(* Logix 5000 project; controller DUNEW2PLC1 vendor 1 type 14 code 221 rev 33.11; software revision 33.00; part 3 of 4 *)
(* tags used below, declared in another part *)
   accel_xy : REAL;   // Tangential acceleration of the winding head in xy-plane
   ACTUATOR_POS : DINT;
   ALL_EOT_GOOD : BOOL;
   APA_IS_VERTICAL : BOOL;
   check_tension_stable : BOOL;   // Check if the tension is stable at the setpoint before moving the winding head
   current_command : REAL;
   current_command_high : REAL;
   current_command_low : REAL;
   ERROR_CODE : DINT;
   gamma : REAL;
   J : REAL;
   LATCH_ACTUATOR_HOMED : BOOL;
   MAS : BOOL;   // Motion Axis Stop
   MASTER_Z_GO : BOOL;
   max_tolerable_tension : REAL;
   MAX_TOLERABLE_Z : REAL;
   MCCD_X_Y_Axis : MOTION_INSTRUCTION;
   MCCD_X_Y_Axis1 : MOTION_INSTRUCTION;
   MORE_STATS : BOOL[32];
   MOVE_TYPE : INT;   // 0 = No Move 1 = XY JOG 2 = XY Plane Move 3 = Z JOG 4 = Z Axis Move 5 = Toggle Latch Actuator 6 = Home the Latch Actuator
   neutral_cv : REAL;
   NEXTSTATE : DINT;
   overtension_timer : TIMER;
   pid_cv_high_limit : REAL;
   pid_cv_low_limit : REAL;
   pid_cv_out : REAL;
   PID_LOOP_TIMER : TIMER;
   pid_loop_timer_bypass : BOOL;
   Safety_Tripped_S : BOOL;
   SetPoint_CV : REAL;
   SetPoint_Override : REAL;
   SetPoint_PV : REAL;   // wire tension from load cell (N)
   SLS_speed : DINT;
   speed_regulator_switch : BOOL;   // This is our "enable safe speed" switch, repurposed to switch the speed regulator
   STATE : DINT;   // CURRENT State Machine State
   tension : ALIAS FOR Local:4:I.Ch01.Data;   // wire tension (N)
   TENSION_CONTROL_OK : BOOL;
   TENSION_ON_SWITCH : BOOL;
   tension_on_switch_delay_on_start : TIMER;
   tension_setpoint : REAL;
   tension_stable_timer : TIMER;
   v_0 : REAL;
   v_xyz : REAL;   // Velocity of winding head in xyz space
   winding_head_pid : PID;
   wire_break_proxy : BOOL;
   X_axis : AXIS_CIP_DRIVE;
   X_Axis_SLS : SAFELY_LIMITED_SPEED;
   X_POSITION : ALIAS FOR POSITION[0,0];
   X_Y : COORDINATE_SYSTEM;
   XY_ACCELERATION : REAL;   // Maximum positive acceleration for position move.
   XY_DECELERATION : REAL;   // Maximum negative acceleration for position move.
   XY_DECELERATION_SLS : REAL;
   xy_regulated_acceleration : REAL;
   xy_regulated_deceleration : REAL;
   XY_SPEED : REAL;   // Maximum velocity for position move.
   XY_SPEED_REQ : REAL;   // XY Requested speed copy of XY_Speed to be used for MCLM and MCCD in MoveXY
   Y_axis : AXIS_CIP_DRIVE;
   Y_POSITION : ALIAS FOR POSITION[0,1];
   Z_ACCELERATION : REAL;
   Z_axis : AXIS_CIP_DRIVE;
   Z_DECELLERATION : REAL;
   Z_FIXED_LATCHED : BOOL;
   Z_POSITION : REAL;
   Z_RETRACTED : BOOL;
   Z_SPEED : REAL;

PROGRAM MoveXY_State_2_3   (* main routine MoveXY *)
VAR
   d_raw : REAL;
   dx : REAL := 0.0039;
   dy : REAL := 0.0017;
   eot_triggered : BOOL;
   k : REAL := 211538.47;
   max_integral : DINT := 1000;
   min_integral : DINT := -1000;
   min_regulated_speed : DINT := 100;
   near_ending : BOOL;   // True if distance to xy-move target is less than the required stopping distance
   near_ending_trigger : BOOL;
   oneshotob : BOOL[32];
   oneshotsb : BOOL[32] := ([2] := 1, [4] := 1, [11] := 1, [12] := 1, [13] := 1, [14] := 1, [15] := 1, [16] := 1, [17] := 1);
   regulated_speed : REAL := 899.9713;
   regulator_loop_timer : TIMER := (PRE := 1);
   speed_set_to_zero : BOOL;
   speed_tension_setpoint : REAL := 8.5;
   starting_x : REAL := -0.0039;
   starting_y : REAL := -0.0017;
   STATE3_IND : BOOL; {access Read Only}
   stopping_distance : REAL;   // Calculate the distance required to perform a jerk-limited stop at the gurrent jerk, acceleration, and speed
   stopping_ratio : REAL := 0.2532453;
   trigger_xy_move : BOOL;
   v_max : REAL := 899.9713;
   x_dist_to_target : REAL := 0.6653;
   X_max_speed : REAL := 825.0; {constant}
   x_time : REAL := 211538.47;
   xy_accel_jerk : DINT := 1500;
   XY_AXIS_STAT : MOTION_INSTRUCTION[32] := ([2].FLAGS := 536870912, [2].DN := 1, [3].FLAGS := 536870912, [3].DN := 1, [4].FLAGS := 33554432, [5].FLAGS := 33554432, [6].FLAGS := 704643072, [6].DN := 1, [6].PC := 1);
   xy_d_alpha : REAL := 1.0;
   xy_d_dt : DINT := 50;
   xy_d_term : REAL;
   xy_d_term_prev : REAL;
   xy_d_timer : TIMER := (PRE := 50);
   xy_decel_jerk : DINT := 2000;
   xy_default_speed : DINT;
   xy_dist_to_target : REAL := 0.66530246;
   xy_dt : DINT := 1;
   xy_error : REAL := 6.0954127;
   xy_error_prev : REAL := 6.0985594;
   xy_i_term : REAL := 900.0352;
   xy_kd : REAL;
   xy_ki : REAL := 300.0;
   xy_kp : REAL;
   xy_p_term : REAL;
   XY_POS_LOCK_STAT : BOOL; {access Read Only}
   y_dist_to_target : REAL := -0.0018;
   Y_max_speed : REAL := 600.0; {constant}
   y_time : REAL := 352941.16;
END_VAR

ROUTINE MoveXY   (* ladder *)
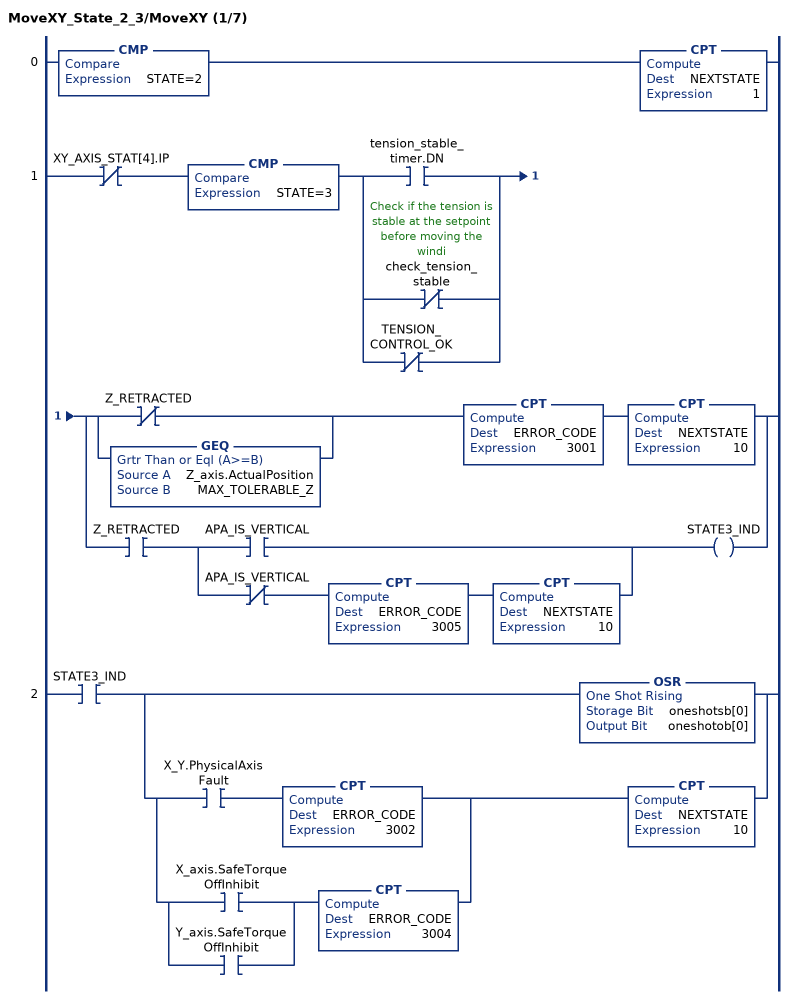
   0: CMP(STATE=2)CPT(NEXTSTATE,1);
   1: XIO(XY_AXIS_STAT[4].IP)CMP(STATE=3)[XIC(tension_stable_timer.DN) ,XIO(check_tension_stable) ,XIO(TENSION_CONTROL_OK) ][[XIO(Z_RETRACTED) ,GEQ(Z_axis.ActualPosition,MAX_TOLERABLE_Z) ] CPT(ERROR_CODE,3001) CPT(NEXTSTATE,10) ,XIC(Z_RETRACTED) [XIC(APA_IS_VERTICAL) ,XIO(APA_IS_VERTICAL) CPT(ERROR_CODE,3005) CPT(NEXTSTATE,10) ] OTE(STATE3_IND) ];
   2: XIC(STATE3_IND)[OSR(oneshotsb[0],oneshotob[0]) ,[XIC(X_Y.PhysicalAxisFault) CPT(ERROR_CODE,3002) ,[XIC(X_axis.SafeTorqueOffInhibit) ,XIC(Y_axis.SafeTorqueOffInhibit) ] CPT(ERROR_CODE,3004) ] CPT(NEXTSTATE,10) ];
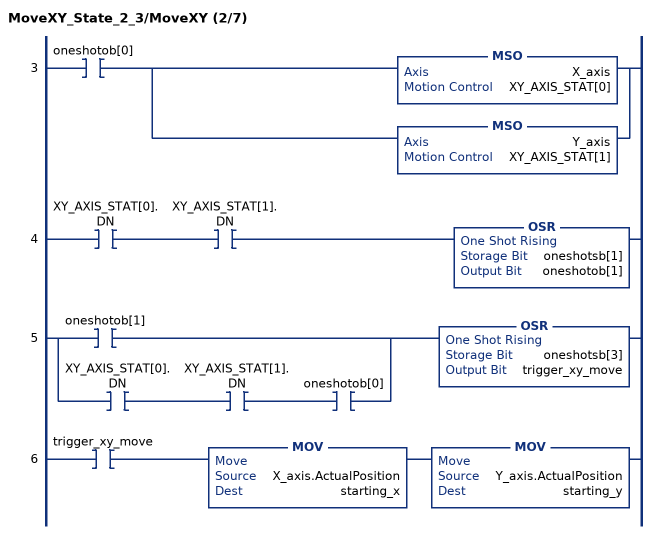
   3: XIC(oneshotob[0])[MSO(X_axis,XY_AXIS_STAT[0]) ,MSO(Y_axis,XY_AXIS_STAT[1]) ];
   4: XIC(XY_AXIS_STAT[0].DN)XIC(XY_AXIS_STAT[1].DN)OSR(oneshotsb[1],oneshotob[1]);
   5: [XIC(oneshotob[1]) ,XIC(XY_AXIS_STAT[0].DN) XIC(XY_AXIS_STAT[1].DN) XIC(oneshotob[0]) ]OSR(oneshotsb[3],trigger_xy_move);
   6: XIC(trigger_xy_move)MOV(X_axis.ActualPosition,starting_x)MOV(Y_axis.ActualPosition,starting_y);
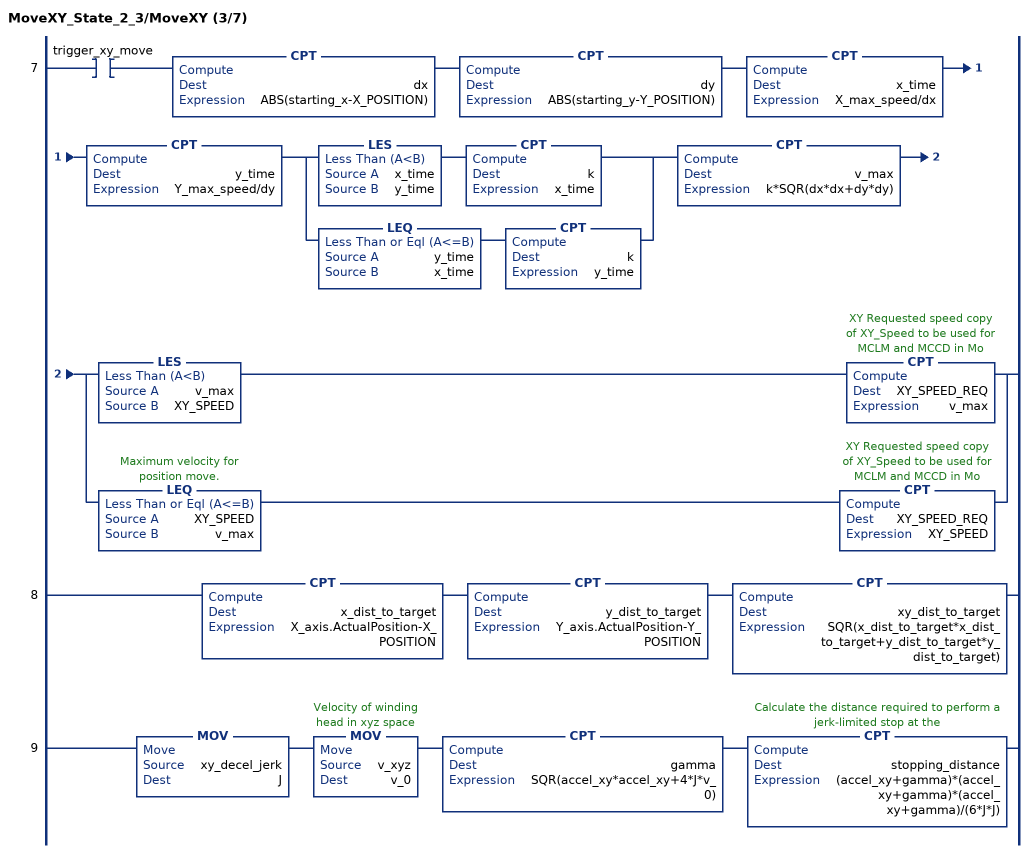
   7: XIC(trigger_xy_move)CPT(dx,ABS(starting_x-X_POSITION))CPT(dy,ABS(starting_y-Y_POSITION))CPT(x_time,X_max_speed/dx)CPT(y_time,Y_max_speed/dy)[LES(x_time,y_time) CPT(k,x_time) ,LEQ(y_time,x_time) CPT(k,y_time) ]CPT(v_max,k*SQR(dx*dx+dy*dy))[LES(v_max,XY_SPEED) CPT(XY_SPEED_REQ,v_max) ,LEQ(XY_SPEED,v_max) CPT(XY_SPEED_REQ,XY_SPEED) ];
   8: CPT(x_dist_to_target,X_axis.ActualPosition-X_POSITION)CPT(y_dist_to_target,Y_axis.ActualPosition-Y_POSITION)CPT(xy_dist_to_target,SQR(x_dist_to_target*x_dist_to_target+y_dist_to_target*y_dist_to_target));
   9: MOV(xy_decel_jerk,J)MOV(v_xyz,v_0)CPT(gamma,SQR(accel_xy*accel_xy+4*J*v_0))CPT(stopping_distance,(accel_xy+gamma)*(accel_xy+gamma)*(accel_xy+gamma)/(6*J*J));
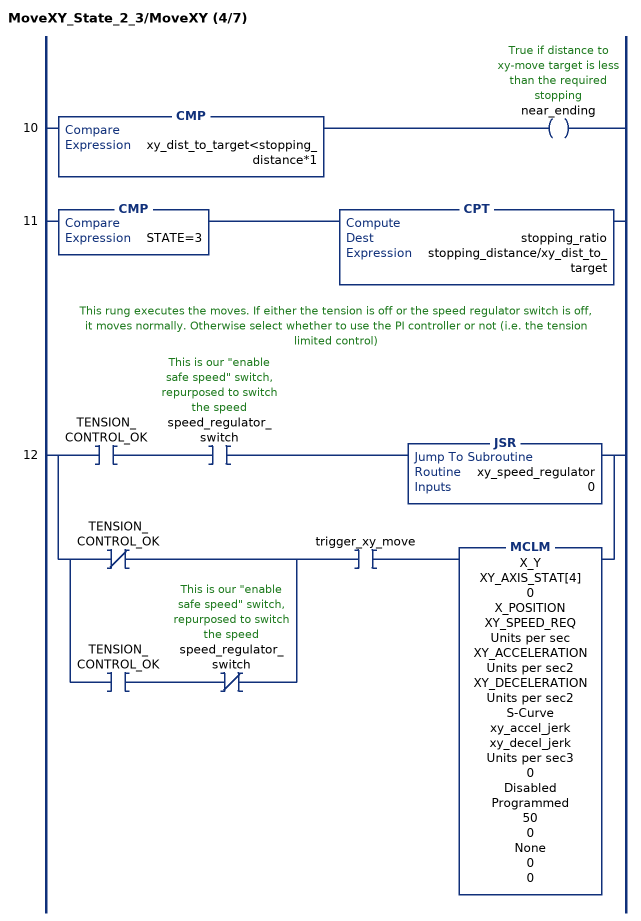
   10: CMP(xy_dist_to_target<stopping_distance*1)OTE(near_ending);
   11: CMP(STATE=3)CPT(stopping_ratio,stopping_distance/xy_dist_to_target);
   // This rung executes the moves. If either the tension is off or the speed regulator switch is off, it moves normally. Otherwise select whether to use the PI controller or not (i.e. the tension limited control)
   12: [XIC(TENSION_CONTROL_OK) XIC(speed_regulator_switch) JSR(xy_speed_regulator,0) ,[XIO(TENSION_CONTROL_OK) ,XIC(TENSION_CONTROL_OK) XIO(speed_regulator_switch) ] XIC(trigger_xy_move) MCLM(X_Y,XY_AXIS_STAT[4],0,X_POSITION,XY_SPEED_REQ,Units per sec,XY_ACCELERATION,Units per sec2,XY_DECELERATION,Units per sec2,S-Curve,xy_accel_jerk,xy_decel_jerk,Units per sec3,0,Disabled,Programmed,50,0,None,0,0) ];
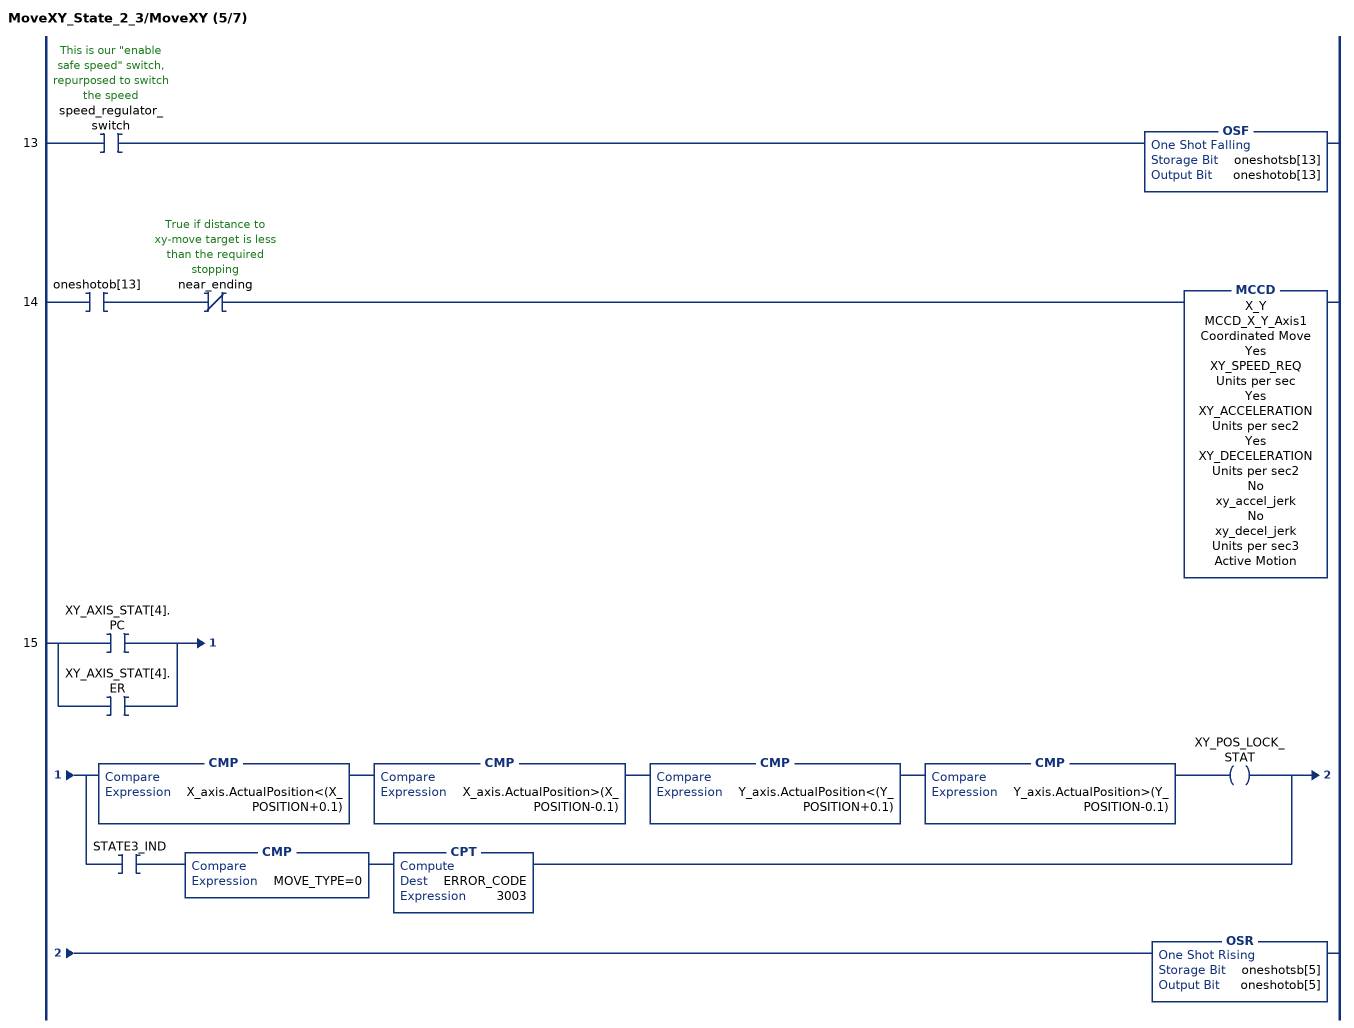
   13: XIC(speed_regulator_switch)OSF(oneshotsb[13],oneshotob[13]);
   14: XIC(oneshotob[13])XIO(near_ending)MCCD(X_Y,MCCD_X_Y_Axis1,Coordinated Move,Yes,XY_SPEED_REQ,Units per sec,Yes,XY_ACCELERATION,Units per sec2,Yes,XY_DECELERATION,Units per sec2,No,xy_accel_jerk,No,xy_decel_jerk,Units per sec3,Active Motion);
   15: [XIC(XY_AXIS_STAT[4].PC) ,XIC(XY_AXIS_STAT[4].ER) ][CMP(X_axis.ActualPosition<(X_POSITION+0.1)) CMP(X_axis.ActualPosition>(X_POSITION-0.1)) CMP(Y_axis.ActualPosition<(Y_POSITION+0.1)) CMP(Y_axis.ActualPosition>(Y_POSITION-0.1)) OTE(XY_POS_LOCK_STAT) ,XIC(STATE3_IND) CMP(MOVE_TYPE=0) CPT(ERROR_CODE,3003) ]OSR(oneshotsb[5],oneshotob[5]);
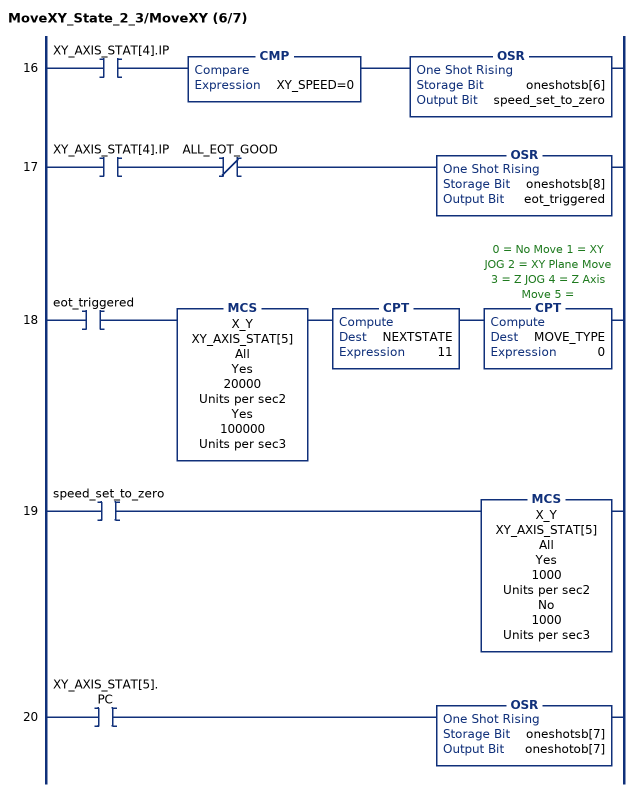
   16: XIC(XY_AXIS_STAT[4].IP)CMP(XY_SPEED=0)OSR(oneshotsb[6],speed_set_to_zero);
   17: XIC(XY_AXIS_STAT[4].IP)XIO(ALL_EOT_GOOD)OSR(oneshotsb[8],eot_triggered);
   18: XIC(eot_triggered)MCS(X_Y,XY_AXIS_STAT[5],All,Yes,20000,Units per sec2,Yes,100000,Units per sec3)CPT(NEXTSTATE,11)CPT(MOVE_TYPE,0);
   19: XIC(speed_set_to_zero)MCS(X_Y,XY_AXIS_STAT[5],All,Yes,1000,Units per sec2,No,1000,Units per sec3);
   20: XIC(XY_AXIS_STAT[5].PC)OSR(oneshotsb[7],oneshotob[7]);
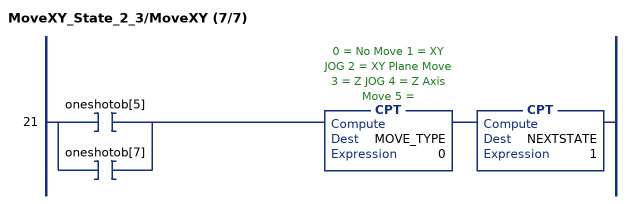
   21: [XIC(oneshotob[5]) ,XIC(oneshotob[7]) ]CPT(MOVE_TYPE,0)CPT(NEXTSTATE,1);
END_ROUTINE

ROUTINE xy_speed_regulator   (* ladder *)
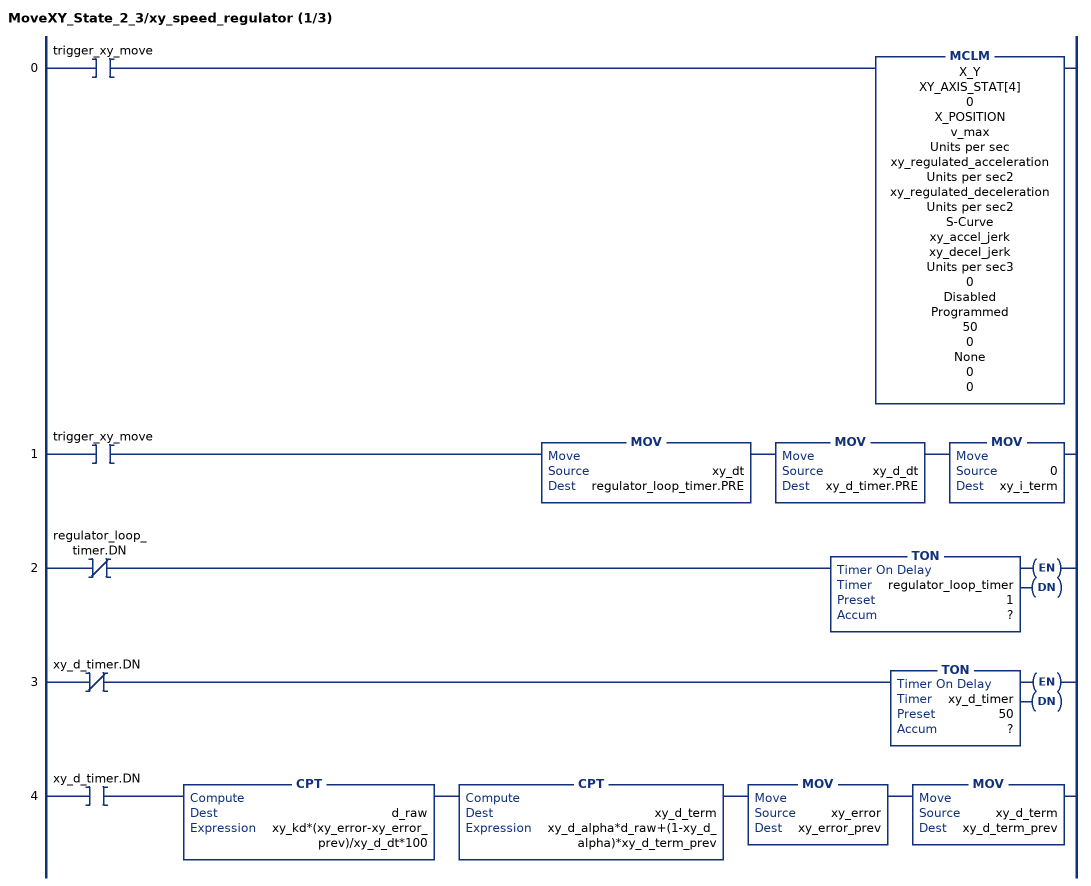
   0: XIC(trigger_xy_move)MCLM(X_Y,XY_AXIS_STAT[4],0,X_POSITION,v_max,Units per sec,xy_regulated_acceleration,Units per sec2,xy_regulated_deceleration,Units per sec2,S-Curve,xy_accel_jerk,xy_decel_jerk,Units per sec3,0,Disabled,Programmed,50,0,None,0,0);
   1: XIC(trigger_xy_move)MOV(xy_dt,regulator_loop_timer.PRE)MOV(xy_d_dt,xy_d_timer.PRE)MOV(0,xy_i_term);
   2: XIO(regulator_loop_timer.DN)TON(regulator_loop_timer,?,?);
   3: XIO(xy_d_timer.DN)TON(xy_d_timer,?,?);
   4: XIC(xy_d_timer.DN)CPT(d_raw,xy_kd*(xy_error-xy_error_prev)/xy_d_dt*100)CPT(xy_d_term,xy_d_alpha*d_raw+(1-xy_d_alpha)*xy_d_term_prev)MOV(xy_error,xy_error_prev)MOV(xy_d_term,xy_d_term_prev);
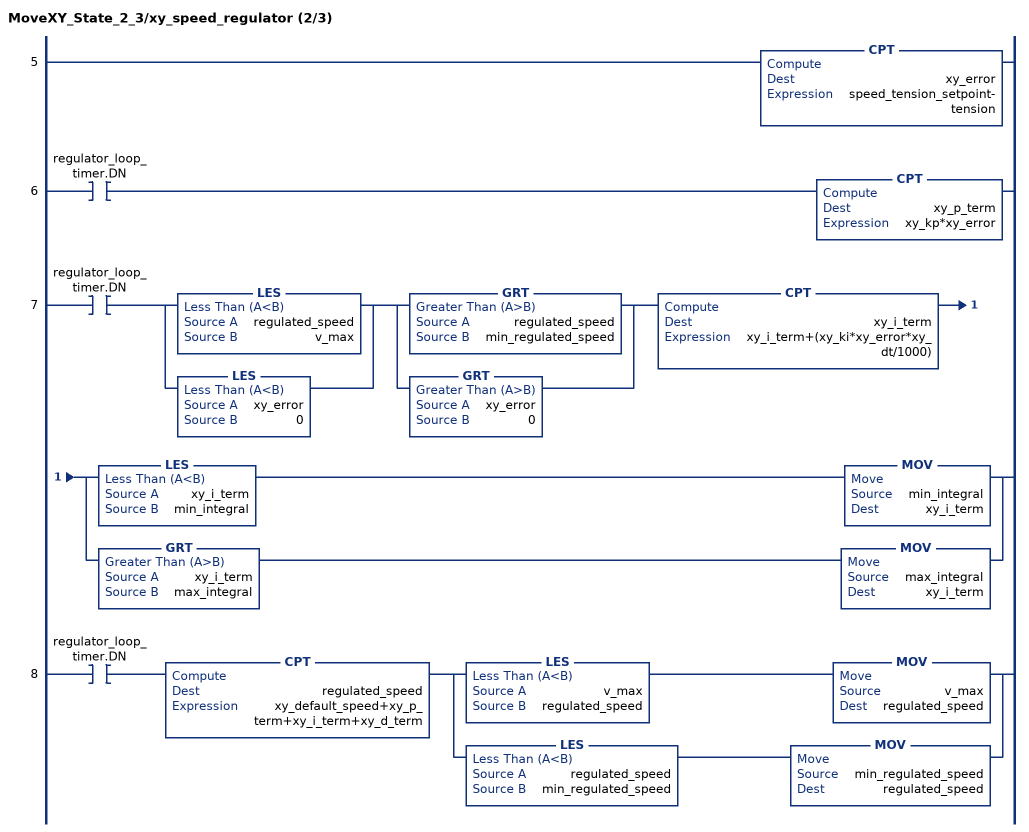
   5: CPT(xy_error,speed_tension_setpoint-tension);
   6: XIC(regulator_loop_timer.DN)CPT(xy_p_term,xy_kp*xy_error);
   7: XIC(regulator_loop_timer.DN)[LES(regulated_speed,v_max) ,LES(xy_error,0) ][GRT(regulated_speed,min_regulated_speed) ,GRT(xy_error,0) ]CPT(xy_i_term,xy_i_term+(xy_ki*xy_error*xy_dt/1000))[LES(xy_i_term,min_integral) MOV(min_integral,xy_i_term) ,GRT(xy_i_term,max_integral) MOV(max_integral,xy_i_term) ];
   8: XIC(regulator_loop_timer.DN)CPT(regulated_speed,xy_default_speed+xy_p_term+xy_i_term+xy_d_term)[LES(v_max,regulated_speed) MOV(v_max,regulated_speed) ,LES(regulated_speed,min_regulated_speed) MOV(min_regulated_speed,regulated_speed) ];
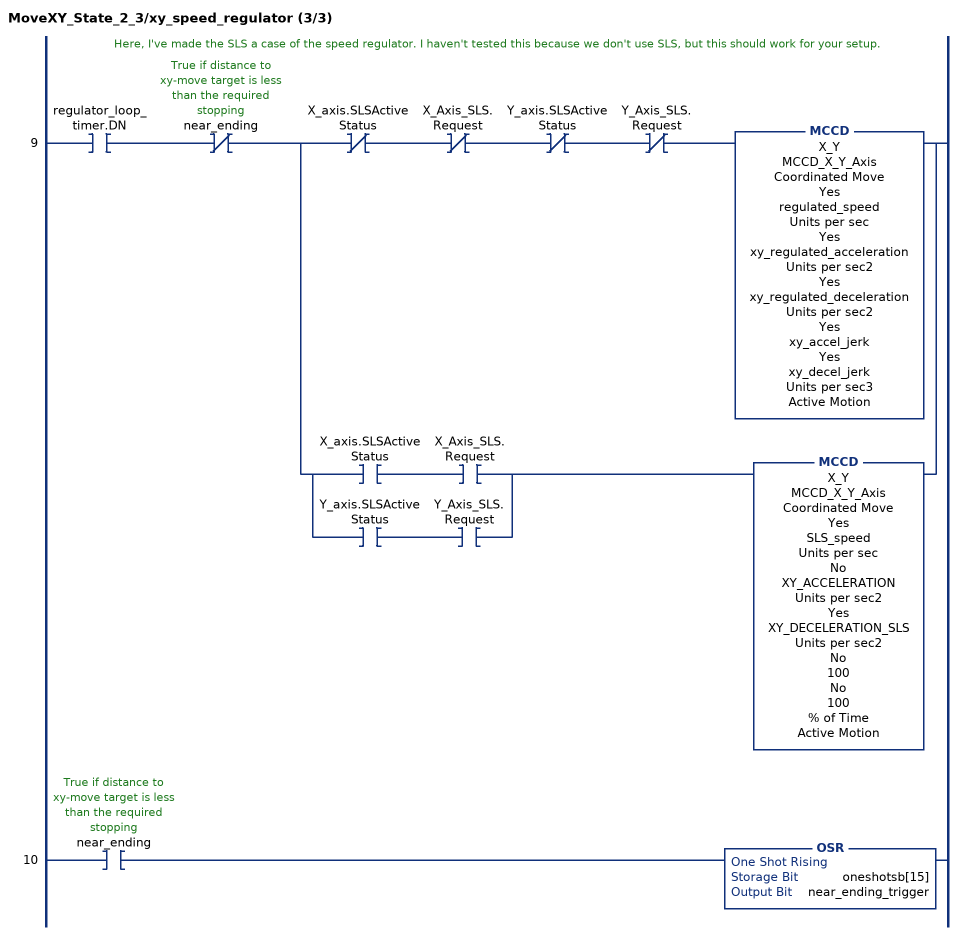
   // Here, I've made the SLS a case of the speed regulator. I haven't tested this because we don't use SLS, but this should work for your setup.
   9: XIC(regulator_loop_timer.DN)XIO(near_ending)[XIO(X_axis.SLSActiveStatus) XIO(X_Axis_SLS.Request) XIO(Y_axis.SLSActiveStatus) XIO(Y_Axis_SLS.Request) MCCD(X_Y,MCCD_X_Y_Axis,Coordinated Move,Yes,regulated_speed,Units per sec,Yes,xy_regulated_acceleration,Units per sec2,Yes,xy_regulated_deceleration,Units per sec2,Yes,xy_accel_jerk,Yes,xy_decel_jerk,Units per sec3,Active Motion) ,[XIC(X_axis.SLSActiveStatus) XIC(X_Axis_SLS.Request) ,XIC(Y_axis.SLSActiveStatus) XIC(Y_Axis_SLS.Request) ] MCCD(X_Y,MCCD_X_Y_Axis,Coordinated Move,Yes,SLS_speed,Units per sec,No,XY_ACCELERATION,Units per sec2,Yes,XY_DECELERATION_SLS,Units per sec2,No,100,No,100,% of Time,Active Motion) ];
   10: XIC(near_ending)OSR(oneshotsb[15],near_ending_trigger);
END_ROUTINE
END_PROGRAM

PROGRAM MoveZ_State_4_5   (* main routine MoveZ *)
VAR
   error_suppress : BOOL;
   oneshotob : BOOL[32]; {access Read Only}
   oneshotsb : BOOL[32] := ([0] := 1, [1] := 1, [2] := 1, [9] := 1, [26] := 1, [28] := 1, [29] := 1, [30] := 1, [31] := 1); {access Read Only}
   STATE5_IND : BOOL; {access Read Only}
   z_accel_jerk : DINT := 800;
   Z_AXIS_STAT : MOTION_INSTRUCTION[32] := ([0].FLAGS := 33554432, [1].FLAGS := 33554432, [2].FLAGS := 33554432, [4].FLAGS := 33554432, [5].FLAGS := 33554432, [6].FLAGS := 33554432, [7].FLAGS := 33554432, [8].FLAGS := 33554432, [9].FLAGS := 536870912, [9].DN := 1); {access Read Only}
   z_decel_jerk : DINT := 1600;
   Z_POS_LOCK_STAT : BOOL; {access Read Only}
END_VAR

ROUTINE MoveZ   (* ladder *)
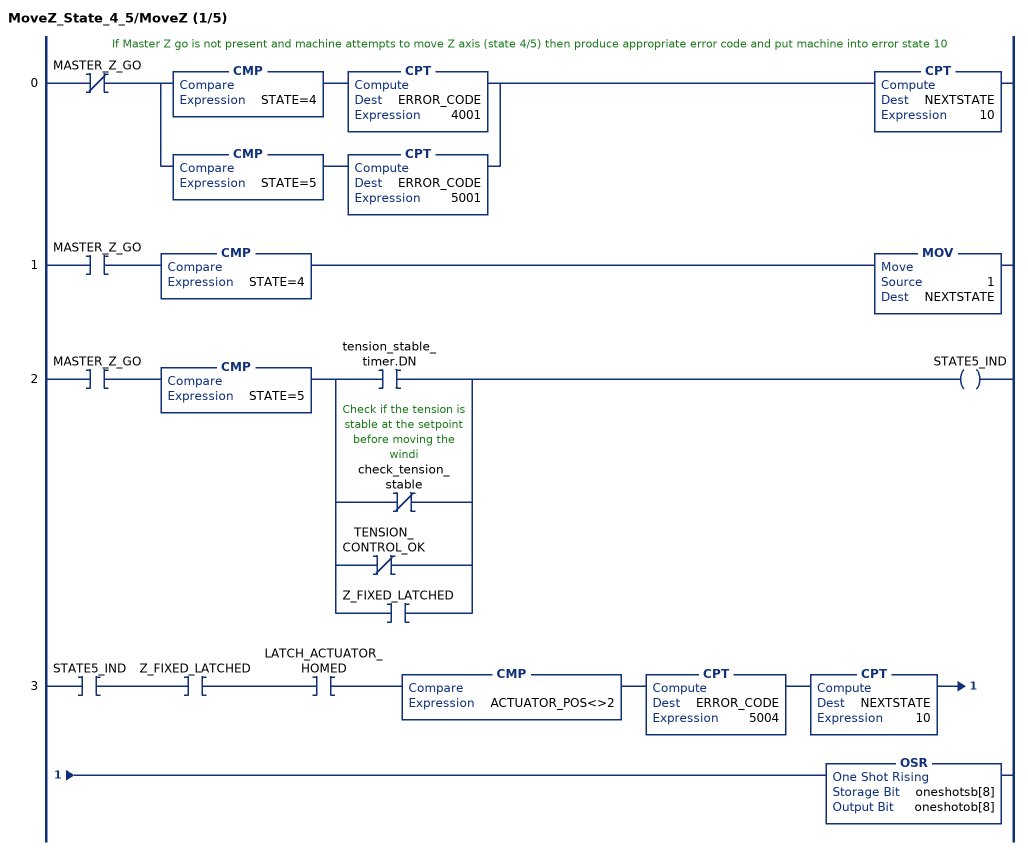
   // If Master Z go is not present and machine attempts to move Z axis (state 4/5) then produce appropriate error code and put machine into error state 10
   0: XIO(MASTER_Z_GO)[CMP(STATE=4) CPT(ERROR_CODE,4001) ,CMP(STATE=5) CPT(ERROR_CODE,5001) ]CPT(NEXTSTATE,10);
   1: XIC(MASTER_Z_GO)CMP(STATE=4)MOV(1,NEXTSTATE);
   2: XIC(MASTER_Z_GO)CMP(STATE=5)[XIC(tension_stable_timer.DN) ,XIO(check_tension_stable) ,XIO(TENSION_CONTROL_OK) ,XIC(Z_FIXED_LATCHED) ]OTE(STATE5_IND);
   3: XIC(STATE5_IND)XIC(Z_FIXED_LATCHED)XIC(LATCH_ACTUATOR_HOMED)CMP(ACTUATOR_POS<>2)CPT(ERROR_CODE,5004)CPT(NEXTSTATE,10)OSR(oneshotsb[8],oneshotob[8]);
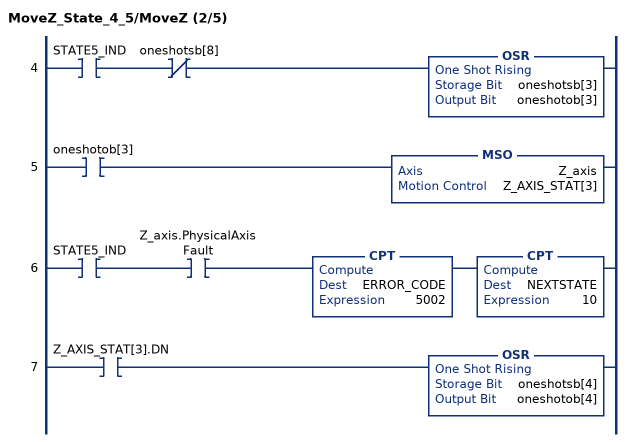
   4: XIC(STATE5_IND)XIO(oneshotsb[8])OSR(oneshotsb[3],oneshotob[3]);
   5: XIC(oneshotob[3])MSO(Z_axis,Z_AXIS_STAT[3]);
   6: XIC(STATE5_IND)XIC(Z_axis.PhysicalAxisFault)CPT(ERROR_CODE,5002)CPT(NEXTSTATE,10);
   7: XIC(Z_AXIS_STAT[3].DN)OSR(oneshotsb[4],oneshotob[4]);
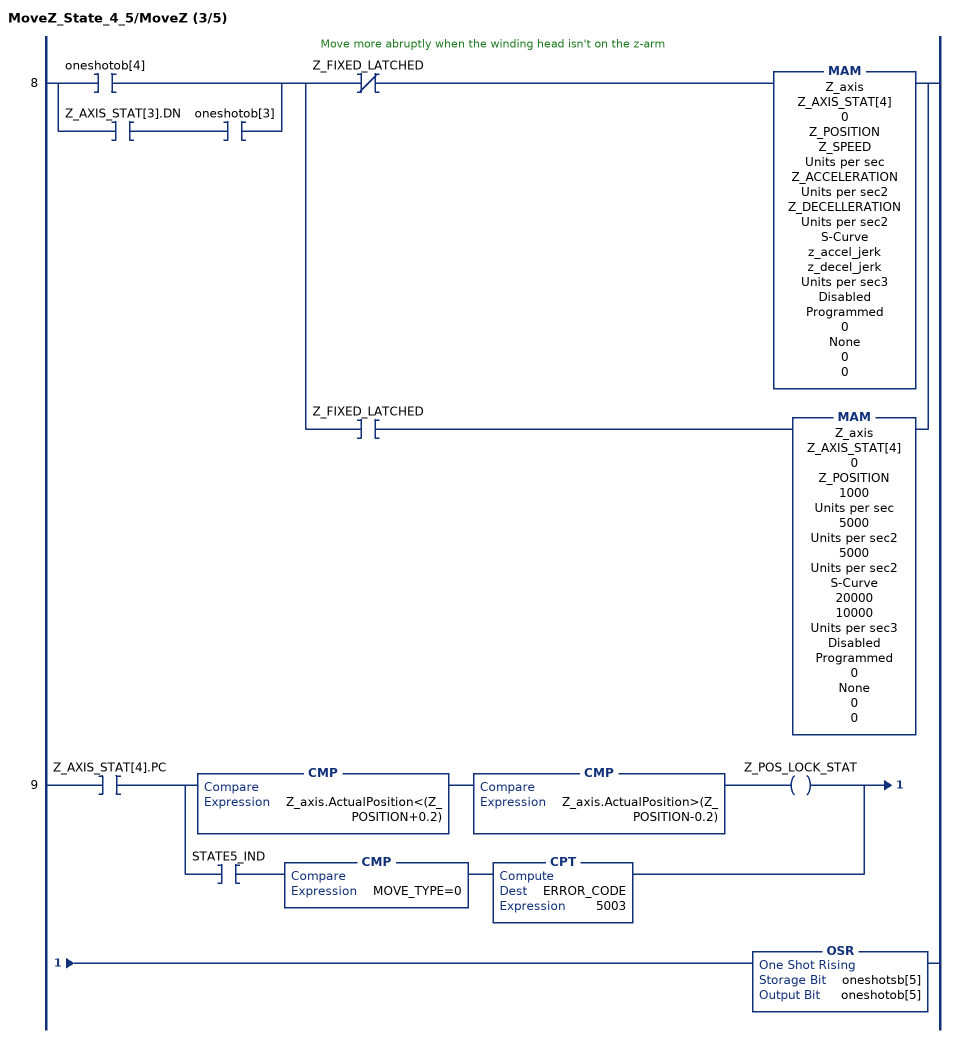
   // Move more abruptly when the winding head isn't on the z-arm
   8: [XIC(oneshotob[4]) ,XIC(Z_AXIS_STAT[3].DN) XIC(oneshotob[3]) ][XIO(Z_FIXED_LATCHED) MAM(Z_axis,Z_AXIS_STAT[4],0,Z_POSITION,Z_SPEED,Units per sec,Z_ACCELERATION,Units per sec2,Z_DECELLERATION,Units per sec2,S-Curve,z_accel_jerk,z_decel_jerk,Units per sec3,Disabled,Programmed,0,None,0,0) ,XIC(Z_FIXED_LATCHED) MAM(Z_axis,Z_AXIS_STAT[4],0,Z_POSITION,1000,Units per sec,5000,Units per sec2,5000,Units per sec2,S-Curve,20000,10000,Units per sec3,Disabled,Programmed,0,None,0,0) ];
   9: XIC(Z_AXIS_STAT[4].PC)[CMP(Z_axis.ActualPosition<(Z_POSITION+0.2)) CMP(Z_axis.ActualPosition>(Z_POSITION-0.2)) OTE(Z_POS_LOCK_STAT) ,XIC(STATE5_IND) CMP(MOVE_TYPE=0) CPT(ERROR_CODE,5003) ]OSR(oneshotsb[5],oneshotob[5]);
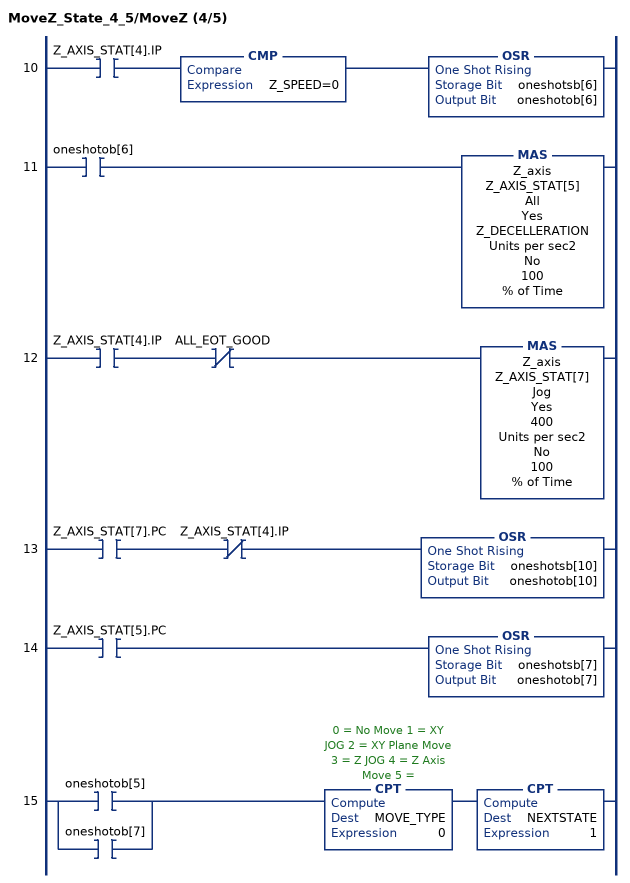
   10: XIC(Z_AXIS_STAT[4].IP)CMP(Z_SPEED=0)OSR(oneshotsb[6],oneshotob[6]);
   11: XIC(oneshotob[6])MAS(Z_axis,Z_AXIS_STAT[5],All,Yes,Z_DECELLERATION,Units per sec2,No,100,% of Time);
   12: XIC(Z_AXIS_STAT[4].IP)XIO(ALL_EOT_GOOD)MAS(Z_axis,Z_AXIS_STAT[7],Jog,Yes,400,Units per sec2,No,100,% of Time);
   13: XIC(Z_AXIS_STAT[7].PC)XIO(Z_AXIS_STAT[4].IP)OSR(oneshotsb[10],oneshotob[10]);
   14: XIC(Z_AXIS_STAT[5].PC)OSR(oneshotsb[7],oneshotob[7]);
   15: [XIC(oneshotob[5]) ,XIC(oneshotob[7]) ]CPT(MOVE_TYPE,0)CPT(NEXTSTATE,1);
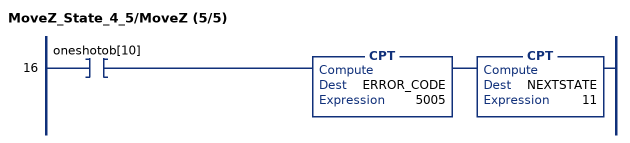
   16: XIC(oneshotob[10])CPT(ERROR_CODE,5005)CPT(NEXTSTATE,11);
END_ROUTINE
END_PROGRAM

PROGRAM PID_Tension_Servo   (* main routine PID_Tension *)
// Using code from Sarah Johnson
VAR
   constant_cv_out : BOOL;
   cv_to_electrocraft : ALIAS FOR Local:5:O.Ch00.Data;
   Enable_tension_motor : ALIAS FOR Local:3:O.Pt03.Data;
   oneshotob : BOOL[32];
   oneshotsb : BOOL[32];
   tension_stable_time : DINT := 200;
   tension_stable_tolerance : REAL := 0.15;
   wire_break_debounce : TIMER := (PRE := 50, ACC := 50, EN := 1, DN := 1);
   wire_break_switch_delay_on_start : TIMER := (PRE := 1000);
END_VAR

ROUTINE PID_Tension   (* ladder *)
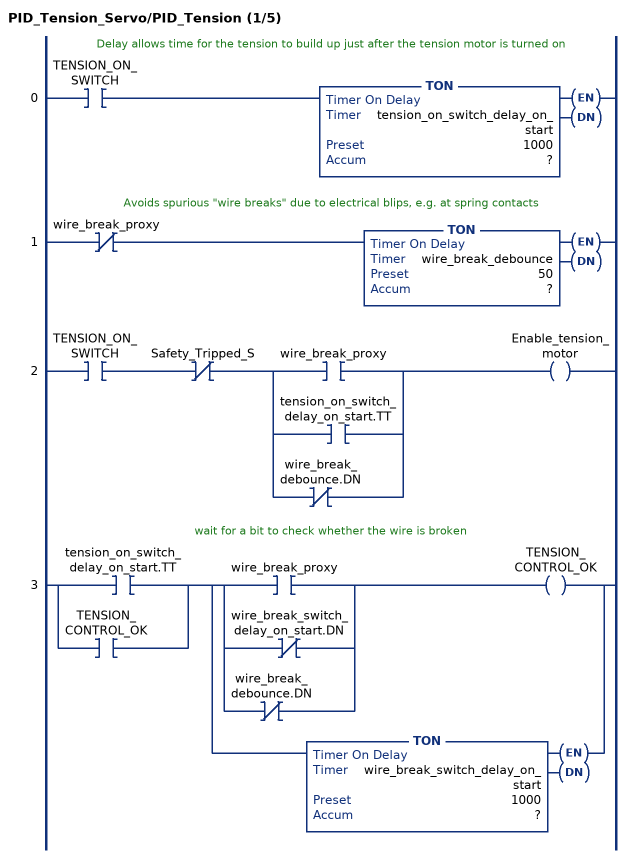
   // Delay allows time for the tension to build up just after the tension motor is turned on
   0: XIC(TENSION_ON_SWITCH)TON(tension_on_switch_delay_on_start,?,?);
   // Avoids spurious "wire breaks" due to electrical blips, e.g. at spring contacts
   1: XIO(wire_break_proxy)TON(wire_break_debounce,?,?);
   2: XIC(TENSION_ON_SWITCH)XIO(Safety_Tripped_S)[XIC(wire_break_proxy) ,XIC(tension_on_switch_delay_on_start.TT) ,XIO(wire_break_debounce.DN) ]OTE(Enable_tension_motor);
   // wait for a bit to check whether the wire is broken
   3: [XIC(tension_on_switch_delay_on_start.TT) ,XIC(TENSION_CONTROL_OK) ][[XIC(wire_break_proxy) ,XIO(wire_break_switch_delay_on_start.DN) ,XIO(wire_break_debounce.DN) ] OTE(TENSION_CONTROL_OK) ,TON(wire_break_switch_delay_on_start,?,?) ];
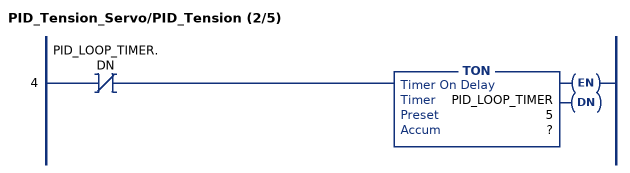
   4: XIO(PID_LOOP_TIMER.DN)TON(PID_LOOP_TIMER,?,?);
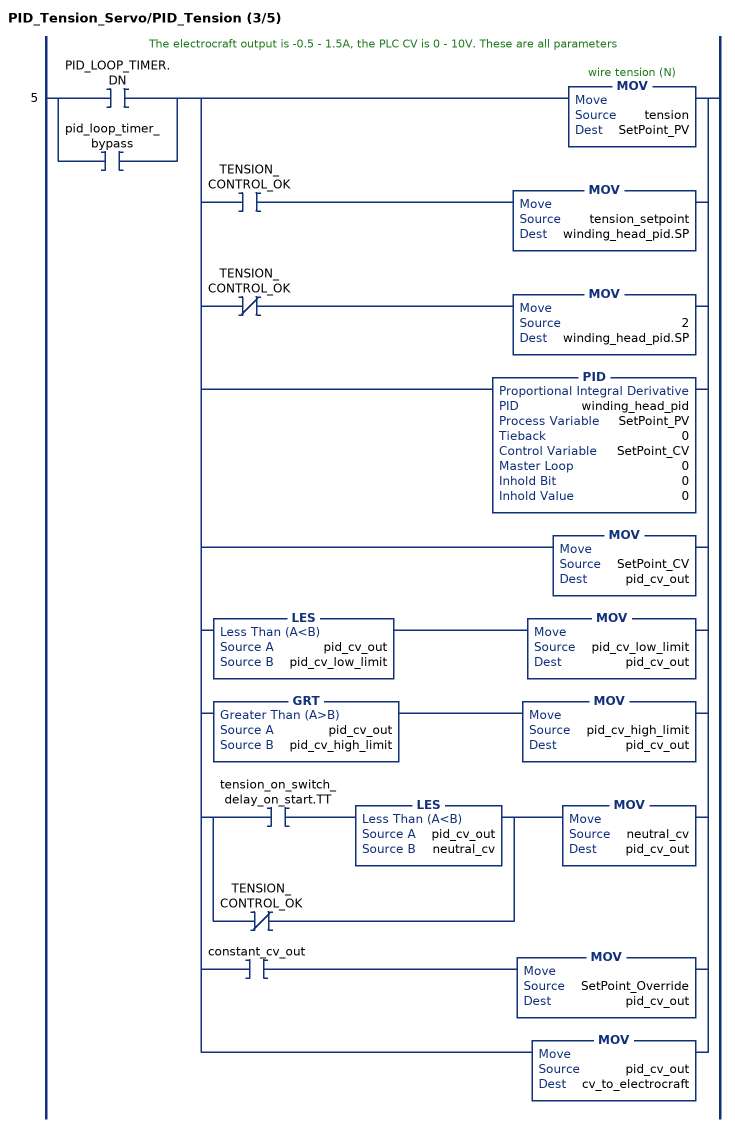
   // The electrocraft output is -0.5 - 1.5A, the PLC CV is 0 - 10V. These are all parameters
   5: [XIC(PID_LOOP_TIMER.DN) ,XIC(pid_loop_timer_bypass) ][MOV(tension,SetPoint_PV) ,XIC(TENSION_CONTROL_OK) MOV(tension_setpoint,winding_head_pid.SP) ,XIO(TENSION_CONTROL_OK) MOV(2,winding_head_pid.SP) ,PID(winding_head_pid,SetPoint_PV,0,SetPoint_CV,0,0,0) ,MOV(SetPoint_CV,pid_cv_out) ,LES(pid_cv_out,pid_cv_low_limit) MOV(pid_cv_low_limit,pid_cv_out) ,GRT(pid_cv_out,pid_cv_high_limit) MOV(pid_cv_high_limit,pid_cv_out) ,[XIC(tension_on_switch_delay_on_start.TT) LES(pid_cv_out,neutral_cv) ,XIO(TENSION_CONTROL_OK) ] MOV(neutral_cv,pid_cv_out) ,XIC(constant_cv_out) MOV(SetPoint_Override,pid_cv_out) ,MOV(pid_cv_out,cv_to_electrocraft) ];
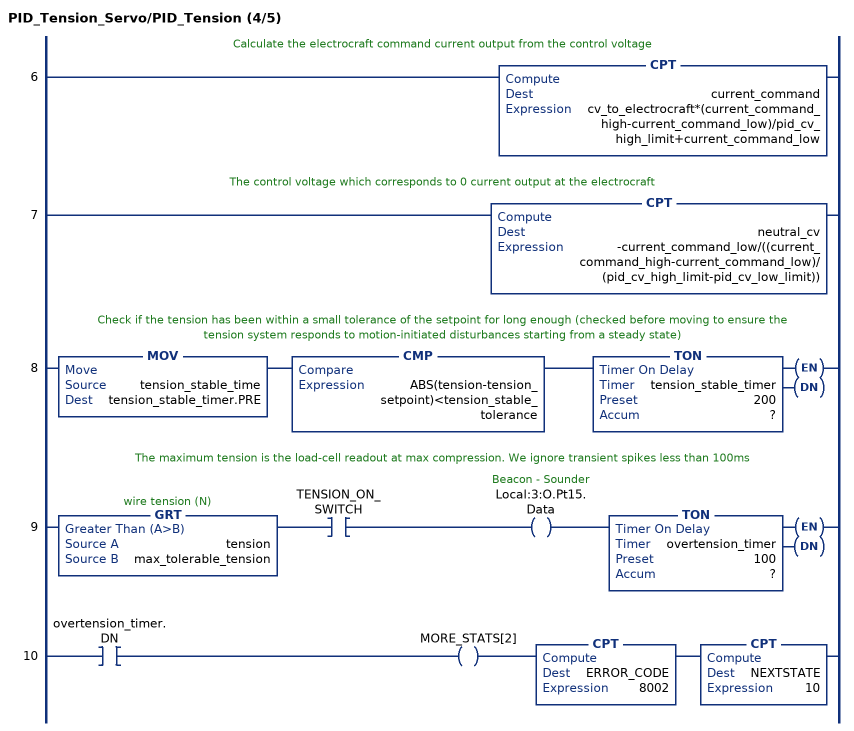
   // Calculate the electrocraft command current output from the control voltage
   6: CPT(current_command,cv_to_electrocraft*(current_command_high-current_command_low)/pid_cv_high_limit+current_command_low);
   // The control voltage which corresponds to 0 current output at the electrocraft
   7: CPT(neutral_cv,-current_command_low/((current_command_high-current_command_low)/(pid_cv_high_limit-pid_cv_low_limit)));
   // Check if the tension has been within a small tolerance of the setpoint for long enough (checked before moving to ensure the tension system responds to motion-initiated disturbances starting from a steady state)
   8: MOV(tension_stable_time,tension_stable_timer.PRE)CMP(ABS(tension-tension_setpoint)<tension_stable_tolerance)TON(tension_stable_timer,?,?);
   // The maximum tension is the load-cell readout at max compression. We ignore transient spikes less than 100ms
   9: GRT(tension,max_tolerable_tension)XIC(TENSION_ON_SWITCH)OTE(Local:3:O.Pt15.Data)TON(overtension_timer,?,?);
   10: XIC(overtension_timer.DN)OTE(MORE_STATS[2])CPT(ERROR_CODE,8002)CPT(NEXTSTATE,10);
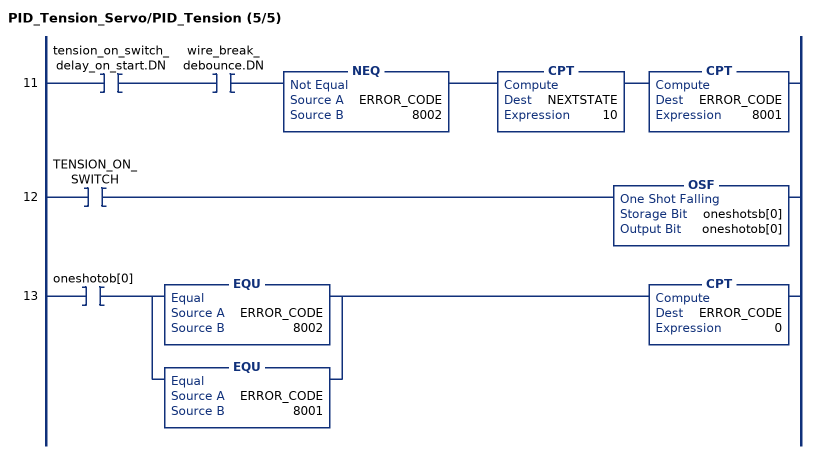
   11: XIC(tension_on_switch_delay_on_start.DN)XIC(wire_break_debounce.DN)NEQ(ERROR_CODE,8002)CPT(NEXTSTATE,10)CPT(ERROR_CODE,8001);
   12: XIC(TENSION_ON_SWITCH)OSF(oneshotsb[0],oneshotob[0]);
   13: XIC(oneshotob[0])[EQU(ERROR_CODE,8002) ,EQU(ERROR_CODE,8001) ]CPT(ERROR_CODE,0);
END_ROUTINE
END_PROGRAM
